FUNCTION_BLOCK ConvSync (* Conveyors synchronization *)
  (* Standard: 61499-2 *)
  (* Version 0.2, 2003-12-05, JHC, Rockwell Automation, Renamed from NEWCOMPFB. *)
  (* Version 0.1, 2002-01-08, JHC, Rockwell Automation, Added DLY FB as example. *)
  (* Version 0.0, 2000-05-27, JHC, Rockwell Automation *)
  (* Compiler header: package fb.rt.template; import fb.rt.mva.*; import fb.rt.compare.*; import fb.rt.events.*; import fb.rt.math.*; *)
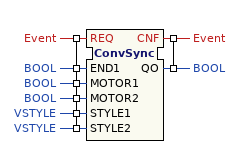
  EVENT_INPUT
    REQ WITH END1, MOTOR1, MOTOR2, STYLE2, STYLE1; (* Normal Execution Request *)
  END_EVENT
  EVENT_OUTPUT
    CNF WITH QO; (* Execution Confirmation *)
  END_EVENT
  VAR_INPUT
    END1 : BOOL; (* Input event qualifier *)
    MOTOR1 : BOOL;
    MOTOR2 : BOOL;
    STYLE1 : VSTYLE := NONE; (* Workpiece style for the curr conv *)
    STYLE2 : VSTYLE := NONE; (* Workpiece style for the next conv *)
  END_VAR
  VAR_OUTPUT
    QO : BOOL; (* Output event qualifier *)
  END_VAR
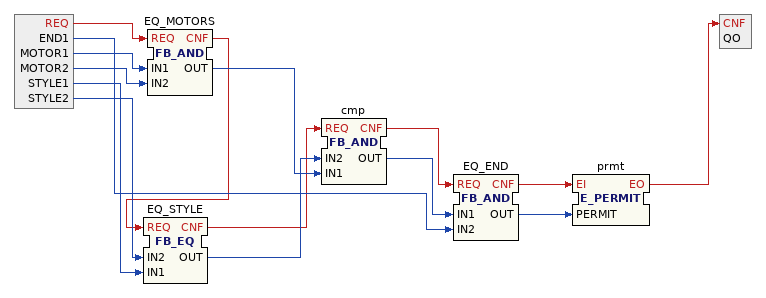
  FBS
    EQ_MOTORS : FB_AND;
    EQ_STYLE : FB_EQ;
    cmp : FB_AND;
    EQ_END : FB_AND;
    prmt : E_PERMIT;
  END_FBS
  EVENT_CONNECTIONS
    REQ TO EQ_MOTORS.REQ;
    EQ_MOTORS.CNF TO EQ_STYLE.REQ;
    EQ_STYLE.CNF TO cmp.REQ;
    cmp.CNF TO EQ_END.REQ;
    EQ_END.CNF TO prmt.EI;
    prmt.EO TO CNF;
  END_CONNECTIONS
  DATA_CONNECTIONS
    MOTOR1 TO EQ_MOTORS.IN1;
    MOTOR2 TO EQ_MOTORS.IN2;
    STYLE2 TO EQ_STYLE.IN2;
    EQ_STYLE.OUT TO cmp.IN2;
    EQ_MOTORS.OUT TO cmp.IN1;
    cmp.OUT TO EQ_END.IN1;
    END1 TO EQ_END.IN2;
    STYLE1 TO EQ_STYLE.IN1;
    EQ_END.OUT TO prmt.PERMIT;
  END_CONNECTIONS
END_FUNCTION_BLOCK
